(* CoDeSys 2.3 export: STRESULTOFMODBUSSLAVESCAN.EXP *)

(* Data type *)
TYPE stResultOfModbusSlaveScan :
STRUCT
	eModbusfunction: MODBUS_FUNCTIONS;
	iModbusAdress: INT;
	wValue: WORD;
	eModbusError: MODBUS_ERRORS;
END_STRUCT
END_TYPE
